// TwinCAT 3 PLC project PlcAppExamples
// Title: PlcAppExamples
// Company: Vortex.Library
// ProjectVersion: 0.6.0.913
// ProgramVersion: 3.1.4024.12
// libraries:
//   Tc2_Standard, * (Beckhoff Automation GmbH)
//   Tc2_System, * (Beckhoff Automation GmbH)
//   Tc3_Module, * (Beckhoff Automation GmbH)
//   TcoCore, 0.6.0.913 (Vortex.Library)
//   TcoPneumatics, 0.6.0.913 (Vortex.Library)
// project tree:
//   / PlcTask.TcTTO
//   POUs/Context/CorleoneKids/ Constanzia_Object.TcPOU, Frederico_Object.TcPOU, Michael_Object.TcPOU, Santino_Object.TcPOU, Thomas_Object.TcPOU
//   POUs/Context/Leaves/ AKid_Object.TcPOU
//   POUs/Context/ VitoCorleone_Context.TcPOU
//   POUs/NonFrameworkUse/ NF_Logic.TcPOU, NF_MAIN.TcPOU
//   POUs/Object/ Horse_Object.TcPOU, Killer_Object.TcPOU, Woltz_Object.TcPOU, Person_Object.TcPOU
//   POUs/Sequencer/ fbAwait.TcPOU, MakeAnOfferThatCantBeRefused.TcPOU, ST_01_Components.TcPOU, ST_01_Context.TcPOU, ST_01_Ground.TcPOU, ST_01_Automat.TcPOU, ST_01_IO.TcGVL
//   POUs/Task/ AskForTheFavor_Task.TcPOU, Kill_Task.TcPOU
//   POUs/Tutorial/101_Color_Sequencer/ ColorSequencer.TcPOU, Color_Example.TcPOU, stColors.TcDUT
//   POUs/Tutorial/201/ InvokingTasks.TcPOU
//   POUs/Tutorial/301/ FastCounter.TcPOU, SlowCounter.TcPOU, TaskExecution.TcPOU
//   POUs/Tutorial/401/ fbPiston.TcPOU, fbPistonMoveTask.TcPOU, IPistonGripper.TcIO, IPistonHorizontal.TcIO, IPistonVertical.TcIO
//   POUs/Tutorial/401/POUs/ Station001.TcPOU, Station001_Components.TcPOU, Station001_Sequencer.TcPOU
//   POUs/Tutorial/ MAIN_PRG.TcPOU, TcOpenTutorial.TcPOU
// real-time tasks:
//   TASK PlcTask: cycle T#10ms, priority 20, ADS port 350

CONFIGURATION PlcAppExamples
    RESOURCE PLC ON TwinCAT3
        TASK PlcTask(INTERVAL := T#10ms, PRIORITY := 20);
        PROGRAM MAIN_PRG WITH PlcTask : MAIN_PRG;
        PROGRAM NF_MAIN WITH PlcTask : NF_MAIN;
    END_RESOURCE
END_CONFIGURATION

// ---- POUs/Tutorial/101_Color_Sequencer/stColors.TcDUT
TYPE stColors :
STRUCT
    _lightR_IsOn : BOOL;
    _lightG_IsOn : BOOL;
    _lightB_IsOn : BOOL;
    _lightR_SwitchOn : BOOL;
    _lightG_SwitchOn : BOOL;
    _lightB_SwitchOn : BOOL;
    _luminosityMin : REAL;
    _luminosity : REAL;
    _luminosityMax : REAL;
END_STRUCT
END_TYPE

// ---- POUs/Sequencer/ST_01_IO.TcGVL
{attribute 'qualified_only'}
VAR_GLOBAL
    INs AT %I* : ARRAY[0..15] OF BOOL;
    OUTs AT %Q* : ARRAY[0..15] OF BOOL;
END_VAR

// ---- POUs/Tutorial/401/IPistonGripper.TcIO
INTERFACE IPistonGripper

METHOD Close : TcoCore.ITcoTaskStatus
END_METHOD

METHOD Open : TcoCore.ITcoTaskStatus
END_METHOD

END_INTERFACE

// ---- POUs/Tutorial/401/IPistonHorizontal.TcIO
INTERFACE IPistonHorizontal

METHOD MoveLeft : TcoCore.ITcoTaskStatus
END_METHOD

METHOD MoveRight : TcoCore.ITcoTaskStatus
END_METHOD

END_INTERFACE

// ---- POUs/Tutorial/401/IPistonVertical.TcIO
INTERFACE IPistonVertical

METHOD MoveDown : TcoCore.ITcoTaskStatus
END_METHOD

METHOD MoveUp : TcoCore.ITcoTaskStatus
END_METHOD

END_INTERFACE

// ---- POUs/Tutorial/MAIN_PRG.TcPOU
PROGRAM MAIN_PRG
VAR
    _pneuMan : ST_01_Context;
    _donCorleone : VitoCorleone_Context;
    _Jack_Woltz : Woltz_Object(_Jack_Woltz);
    _TcOpenTutorial : TcOpenTutorial;
END_VAR

_pneuMan.Run();
_donCorleone.Run();
_TcOpenTutorial.Run();

END_PROGRAM

// ---- POUs/Sequencer/ST_01_Context.TcPOU
// This is an example of a simple pneumatic manipulator 2 pistons 1 gripper.
// Note that this block is extended by 'TcoCore.TcoContext'.
FUNCTION_BLOCK ST_01_Context EXTENDS TcoCore.TcoContext
VAR
    // Ground position sequence
    _groundSequcence : ST_01_Ground(THIS^, eRestoreMode.None);
    // Automat mode sequence
    _automatSequence : ST_01_Automat(THIS^, eRestoreMode.None);
    // Task to execute _groundSequence
    _groundTask : TcoCore.TcoTask(THIS^);
    // Task to execute _automatSequence
    _automatTask : TcoCore.TcoTask(THIS^);
END_VAR

(*~
    <docu>
        <summary>
            Main method of the TcoContext. This is the entry point of any control logic that belongs to this context.
            The call of this method is ensured by calling the <c>InstanceName.Run()</c> method, and it must not be called explicitly.
            This method is abstract, and it must be overriden in inherited block.
        </summary>
    </docu>
~*)
METHOD PROTECTED Main
IF (_groundTask.Execute()) THEN
    _groundSequcence.Run();
    _groundTask.DoneWhen(_groundSequcence._currentStep.ID = 400);
END_IF;

IF (_groundSequcence._currentStep.ID = 400 AND_THEN _automatTask.Execute()) THEN
    _automatSequence.Run();
END_IF;
END_METHOD

END_FUNCTION_BLOCK

// ---- POUs/Sequencer/ST_01_Ground.TcPOU
FUNCTION_BLOCK ST_01_Ground EXTENDS TcoCore.TcoSequencer
VAR
    _components : ST_01_Components(THIS^);
    _await : fbAwait;
END_VAR

(*~
    <docu>
        <summary>
            Main method of the sequener. Custom code needs to be placed here, calling of the methods Open() at the beggining and Close() at the end is ensured by calling the InstanceName.Run() method.
            This method is abstract, so each derived type has to implement its own implementation of this method.
        </summary>
    </docu>
~*)
METHOD PROTECTED Main : BOOL
IF (Step(inStepID := 100, inEnabled := TRUE, inStepDescription := 'VERTICAL CYLINDER UP')) THEN
    //-------------------------------------------------------------
    THIS^.StepCompleteWhen(THIS^._components._vertical.MoveToHome().Done OR _await.Sometime());
    //-------------------------------------------------------------
END_IF

IF (Step(inStepID := 200, inEnabled := TRUE, inStepDescription := 'HORIZONTAL CYLINDER HOME')) THEN
    //-------------------------------------------------------------
    THIS^.StepCompleteWhen(THIS^._components._horizontal.MoveToHome().Done OR _await.Sometime());
    //-------------------------------------------------------------
END_IF

IF (Step(inStepID := 300, inEnabled := TRUE, inStepDescription := 'OPEN GRIPPER')) THEN
    //-------------------------------------------------------------
    THIS^.StepCompleteWhen(THIS^._components._gripper.MoveToHome().Done OR _await.Sometime());
    //-------------------------------------------------------------
END_IF

IF (Step(inStepID := 400, inEnabled := TRUE, inStepDescription := 'CLOSE SEQUENCE')) THEN
    //-------------------------------------------------------------
    //-------------------------------------------------------------
END_IF
END_METHOD

END_FUNCTION_BLOCK

// ---- POUs/Sequencer/ST_01_Components.TcPOU
FUNCTION_BLOCK ST_01_Components EXTENDS TcoCore.TcoObject
VAR
    _horizontal : TcoPneumatics.TcoCylinder(THIS^);
    _vertical : TcoPneumatics.TcoCylinder(THIS^);
    _gripper : TcoPneumatics.TcoCylinder(THIS^);
END_VAR

_horizontal(inoAtHomePos := ST_01_IO.INs[0],
    inoAtWorkPos := ST_01_IO.INs[1],
    inoToHomePos := ST_01_IO.OUTs[0],
    inoToWorkPos := ST_01_IO.OUTs[1]);

_vertical(inoAtHomePos := ST_01_IO.INs[2],
    inoAtWorkPos := ST_01_IO.INs[3],
    inoToHomePos := ST_01_IO.OUTs[2],
    inoToWorkPos := ST_01_IO.OUTs[3]);

_gripper(inoAtHomePos := ST_01_IO.INs[4],
    inoAtWorkPos := ST_01_IO.INs[5],
    inoToHomePos := ST_01_IO.OUTs[4],
    inoToWorkPos := ST_01_IO.OUTs[5]);

END_FUNCTION_BLOCK

// ---- POUs/Sequencer/fbAwait.TcPOU
FUNCTION_BLOCK fbAwait
VAR
    Timer : Tc2_Standard.TON;
END_VAR

METHOD Delay : BOOL
VAR_INPUT
    Timespan : TIME;
END_VAR
Timer(IN := TRUE, PT := Timespan);

IF Timer.Q THEN
    Timer(IN := FALSE, PT := T#0S);
    Delay := TRUE;
ELSE
    Delay := FALSE;
END_IF
END_METHOD

METHOD Sometime : BOOL
VAR_INPUT
END_VAR
Sometime := Delay(T#1S);
END_METHOD

END_FUNCTION_BLOCK

// ---- POUs/Sequencer/ST_01_Automat.TcPOU
FUNCTION_BLOCK ST_01_Automat EXTENDS TcoCore.TcoSequencer
VAR
    _components : ST_01_Components(THIS^);
    _await : fbAwait;
END_VAR

(*~
    <docu>
        <summary>
            Main method of the sequener. Custom code needs to be placed here, calling of the methods Open() at the beggining and Close() at the end is ensured by calling the InstanceName.Run() method.
            This method is abstract, so each derived type has to implement its own implementation of this method.
        </summary>
    </docu>
~*)
METHOD PROTECTED Main : BOOL
_components();

IF (Step(inStepID := 100, inEnabled := TRUE, inStepDescription := 'GROUND')) THEN
    //-------------------------------------------------------------
    THIS^.StepCompleteWhen(_await.Sometime() OR
            (THIS^._components._vertical.MoveToHome().Done AND_THEN
            THIS^._components._horizontal.MoveToHome().Done AND_THEN
            THIS^._components._gripper.MoveToHome().Done));
    //-------------------------------------------------------------
END_IF

IF (Step(inStepID := 200, inEnabled := TRUE, inStepDescription := 'VERTICAL CYLINDER DOWN TO LOAD')) THEN
    //-------------------------------------------------------------
    THIS^.StepCompleteWhen(_await.Sometime() OR (THIS^._components._vertical.MoveToWork().Done));
    //-------------------------------------------------------------
END_IF

IF (Step(inStepID := 300, inEnabled := TRUE, inStepDescription := 'CLOSE GRIPPER')) THEN
    //-------------------------------------------------------------
    THIS^.StepCompleteWhen(_await.Sometime() OR (THIS^._components._gripper.MoveToWork().Done));
    //-------------------------------------------------------------
END_IF

IF (Step(inStepID := 400, inEnabled := TRUE, inStepDescription := 'VERTICAL CYLINDER UP')) THEN
    //-------------------------------------------------------------
    THIS^.StepCompleteWhen(_await.Sometime() OR (THIS^._components._vertical.MoveToHome().Done));
    //-------------------------------------------------------------
END_IF

IF (Step(inStepID := 500, inEnabled := TRUE, inStepDescription := 'HORIZONTAL TO UNLOAD POSITION')) THEN
    //-------------------------------------------------------------
    THIS^.StepCompleteWhen(_await.Sometime() OR (THIS^._components._horizontal.MoveToWork().Done));
    //-------------------------------------------------------------
END_IF

IF (Step(inStepID := 600, inEnabled := TRUE, inStepDescription := 'VERTICAL DOWN TO UNLOAD POSITION')) THEN
    //-------------------------------------------------------------
    THIS^.StepCompleteWhen(_await.Sometime() OR (THIS^._components._vertical.MoveToWork().Done));
    //-------------------------------------------------------------
END_IF

IF (Step(inStepID := 700, inEnabled := TRUE, inStepDescription := 'OPEN GRIPPER')) THEN
    //-------------------------------------------------------------
    THIS^.StepCompleteWhen(_await.Sometime() OR (THIS^._components._gripper.MoveToHome().Done));
    //-------------------------------------------------------------
END_IF

IF (Step(inStepID := 800, inEnabled := TRUE, inStepDescription := 'DONE')) THEN
    //-------------------------------------------------------------
    CompleteSequence();
    //-------------------------------------------------------------
END_IF
END_METHOD

END_FUNCTION_BLOCK

// ---- POUs/Context/VitoCorleone_Context.TcPOU
//--
// <ContextExampleDeclarations>
(*

    THIS EXAMPLE AIMS TO EXPLAIN WHAT CONTEXT AND IDENITY ARE IN A 'TcoOpen' APPLICATION.
    SEE Main() method of this block.

*)
FUNCTION_BLOCK VitoCorleone_Context EXTENDS TcoCore.TcoContext
VAR
    (*
    Each context member object has it 'context' and assigned when instantiated (at birth)
    This is typically done by instantiating the objects with FB_init(ITcoObject) as follows
    These are Don Corleone's children. When you look inside definitions you' find
    Don Corleone's grand-childrend (whole family shares the same context).
*)
    _santino : Santino_Object(THIS^);
    _thomas : Thomas_Object(THIS^);
    _frederico : Frederico_Object(THIS^);
    _michael : Michael_Object(THIS^);
    _costanzia : Constanzia_Object(THIS^);
END_VAR
VAR
    _donCorleoneContext : ITcoContext;
    _isSameContext : BOOL;
    _donCorleoneIdentity : ULINT;
    _isDifferentIndentity : BOOL;
END_VAR
// </ContextExampleDeclarations>
//--
VAR
    _JohnyFontaneCaseDone : BOOL := FALSE;
    _MakeAnOfferThatCantBeRefused : MakeAnOfferThatCantBeRefused(THIS^, eRestoreMode.None);
END_VAR

METHOD JohnyFontaneCase
VAR_INPUT
    Jack_Woltz : REFERENCE TO Woltz_Object;
END_VAR
IF NOT _JohnyFontaneCaseDone THEN
    _MakeAnOfferThatCantBeRefused(Thomas := _thomas, Jack_Woltz := Jack_Woltz, Done => _JohnyFontaneCaseDone);
END_IF;
END_METHOD

(*~
    <docu>
        <summary>
            Main method of the TcoContext. This is the entry point of any control logic that belongs to this context.
            The call of this method is ensured by calling the <c>InstanceName.Run()</c> method, and it must not be called explicitly.
            This method is abstract, and it must be overridden in derived block.
        </summary>
    </docu>
~*)
METHOD PROTECTED Main
//--
// <ContextExampleCode>
(*

                    CONTEXT vs IDENTITY

*)
// In Corleone family they all share the same context that is that of Don Vito Corleone
// Here is the tree of family Corleone
// https://godfather.fandom.com/wiki/Corleone_family
_donCorleoneContext := THIS^.Context;

_isSameContext :=
// Santino
    _donCorleoneContext = THIS^._santino.Context
// Santino's kids
    AND
    (THIS^._santino.Context = THIS^._santino._francesca.Context AND
    THIS^._santino.Context = THIS^._santino._frank.Context AND
    THIS^._santino.Context = THIS^._santino._kathryn.Context AND
    THIS^._santino.Context = THIS^._santino._santino.Context)
// Thomas
    AND
    THIS^._santino.Context = THIS^._thomas.Context
// Thomas' kids
    AND
    (THIS^._thomas.Context = THIS^._thomas._andrew.Context AND
    THIS^._thomas.Context = THIS^._thomas._christina.Context AND
    THIS^._thomas.Context = THIS^._thomas._frank.Context AND
    THIS^._thomas.Context = THIS^._thomas._gianna.Context)
// Frederico
    AND
    THIS^._thomas.Context = THIS^._frederico.Context
// Frederico's kids
    AND
    (THIS^._frederico.Context = THIS^._frederico._fredo.Context)
// Michael
    AND
    THIS^._frederico.Context = THIS^._michael.Context
// Michael's kids
    AND
    (THIS^._michael.Context = THIS^._michael._anthony.Context AND THIS^._michael.Context = THIS^._michael._mary.Context)
// Constanzia
    AND
    THIS^._michael.Context = THIS^._costanzia.Context
// Constanzia's kids
    AND
    (THIS^._costanzia.Context = THIS^._costanzia._michael.Context AND THIS^._costanzia.Context = THIS^._costanzia._victor.Context);
// However each member of the family has different personal identity and that might
// be source of trouble
_donCorleoneIdentity := THIS^.Identity;

_isDifferentIndentity :=
// Santino
    _donCorleoneIdentity <> THIS^._santino.Identity
// Santino's kids
    AND
    (THIS^._santino.Identity <> THIS^._santino._francesca.Identity AND
    THIS^._santino.Identity <> THIS^._santino._frank.Identity AND
    THIS^._santino.Identity <> THIS^._santino._kathryn.Identity AND
    THIS^._santino.Identity <> THIS^._santino._santino.Identity)
// Thomas
    AND
    THIS^._santino.Identity <> THIS^._thomas.Identity
// Thomas' kids
    AND
    (THIS^._thomas.Identity <> THIS^._thomas._andrew.Identity AND
    THIS^._thomas.Identity <> THIS^._thomas._christina.Identity AND
    THIS^._thomas.Identity <> THIS^._thomas._frank.Identity AND
    THIS^._thomas.Identity <> THIS^._thomas._gianna.Identity)
// Frederico
    AND
    THIS^._thomas.Identity <> THIS^._frederico.Identity
// Frederico's kids
    AND
    (THIS^._frederico.Identity <> THIS^._frederico._fredo.Identity)
// Michael
    AND
    THIS^._frederico.Identity <> THIS^._michael.Identity
// Michael's kids
    AND
    (THIS^._michael.Identity <> THIS^._michael._anthony.Identity AND THIS^._michael.Identity <> THIS^._michael._mary.Identity)
// Constanzia
    AND
    THIS^._michael.Identity <> THIS^._costanzia.Identity
// Constanzia's kids
    AND
    (THIS^._costanzia.Identity <> THIS^._costanzia._michael.Identity AND THIS^._costanzia.Identity <> THIS^._costanzia._victor.Identity);
// Once the context is asigned (at birth [instantiated]) it cannot be changed,
// an attempt to change the context will result in vendetta.
// </ContextExampleCode>
//--
JohnyFontaneCase(MAIN_PRG._Jack_Woltz);
END_METHOD

END_FUNCTION_BLOCK

// ---- POUs/Context/CorleoneKids/Santino_Object.TcPOU
FUNCTION_BLOCK Santino_Object EXTENDS TcoCore.TcoObject
VAR
    _francesca : AKid_Object(THIS^);
    _kathryn : AKid_Object(THIS^);
    _frank : AKid_Object(THIS^);
    _santino : AKid_Object(THIS^);
END_VAR

END_FUNCTION_BLOCK

// ---- POUs/Context/Leaves/AKid_Object.TcPOU
FUNCTION_BLOCK AKid_Object EXTENDS TcoCore.TcoObject

END_FUNCTION_BLOCK

// ---- POUs/Context/CorleoneKids/Thomas_Object.TcPOU
FUNCTION_BLOCK Thomas_Object EXTENDS TcoCore.TcoObject
VAR
    _frank : AKid_Object(THIS^);
    _andrew : AKid_Object(THIS^);
    _christina : AKid_Object(THIS^);
    _gianna : AKid_Object(THIS^);
END_VAR
VAR
    _AskForTheFavor : AskForTheFavor_Task(THIS^);
END_VAR

METHOD AskForTheFavor : TcoCore.ITcoTask
VAR_INPUT
    Person_Requested : REFERENCE TO Person_Object;
    RequestedFavor : STRING;
    ReturnFavor : STRING;
END_VAR
_AskForTheFavor(_Person_Requested := Person_Requested, _RequestedFavor := RequestedFavor, _ReturnFavor := ReturnFavor);
AskForTheFavor := _AskForTheFavor;
END_METHOD

END_FUNCTION_BLOCK

// ---- POUs/Task/AskForTheFavor_Task.TcPOU
//--
// <TaskExampleDeclarations>
(*

    This example shows using the 'Tcotask' application. 'TcoTask' is the simplest
    'TcoOpen' coordination primitive.
    In general the body of the task could be devided into the three section:
        1.)	Action
        2.)	Termination condition for the expected behavior.
        3.)	Termination condition for the non-expected behavior.
    The body of the 'Tcotask' needs to be called cyclically. The 'Tcotask' could be then
    invoked from 'outside'. The task of this 'Tcotask' is to ask for the favor
    (in the name of the 'TcoContext' in this example Don Corleone) and offer the return favor.
    Task could end up the expected way in the 'DONE' state if the requested person grant
    the favor or it could end up in the 'ERROR' state if the requested person refuses to grant
    the favor. Each task could be invoked only from the 'READY' state. So if the task enters
    the 'ERROR' state, it cannot be invoked again and has to be restored before. Anyway in this
    example this task is never restored and invoked again as Don Corleone never asks for the
    next favor if the first one was refused.

*)
FUNCTION_BLOCK AskForTheFavor_Task EXTENDS TcoCore.TcoTask
VAR_INPUT
    (*
    'Parameters' of this task are assigned in this example from 'outside' from the
    'upper level' of the hierarchy, where Invoke() method is triggered.
*)
    _Person_Requested : REFERENCE TO Person_Object;
    _RequestedFavor : STRING;
    _ReturnFavor : STRING;
END_VAR
// </TaskExampleDeclarations>
//--

//--
// <TaskBodyExampleCode>
// THIS part needs to be called cyclically.
IF Execute() THEN
    // First section: Action.
    // Meet the right person and interpret the requirements so as a possible return favor.
    _Person_Requested.RequestForTheFavor(_RequestedFavor, _ReturnFavor);
    // Let the person requested to think carefully about the proposition.
    _Person_Requested.ThinkCarefully();
    // Second section: Termination condition for the expected behavior.
    // In the case that the requested person is "smart" and "show the respect" to the
    // 'TcoContext', task finishes in the 'DONE' state and process of the granted the
    // return favor should be started.
    DoneWhen(_Person_Requested.FavorIsGranted());
    // Third section: Termination condition for the non-expected behavior.
    // In the case that the requested person is so self-confident and refuse to grant
    // the favor, task finishes in the 'ERROR' state and automatically the OnTaskError()
    // method is triggered. In this method normally the value of the ReturnFavor is
    // drammatically decreased OR changed to 'Nothing'. Anyway the requested person still
    // have the possibility to grant the favor but under different condition, as he
    // "had to do it the hard way".
    ThrowWhen(_Person_Requested.FavorIsRefused());
END_IF

// </TaskBodyExampleCode>
//--

METHOD PROTECTED OnTaskError
_Person_Requested.ReturnFavor := 'Nothing, and all expenses paid by the recipient.';
END_METHOD

END_FUNCTION_BLOCK

// ---- POUs/Object/Person_Object.TcPOU
FUNCTION_BLOCK Person_Object EXTENDS TcoCore.TcoObject
VAR
    _RequestedFavor : STRING;
    _ReturnFavor : STRING;
    _refuseFavor : BOOL := FALSE;
    _grantFavor : BOOL := FALSE;
END_VAR

METHOD FavorIsGranted : BOOL
VAR_INPUT
END_VAR
FavorIsGranted := _grantFavor;
END_METHOD

METHOD FavorIsRefused : BOOL
VAR_INPUT
END_VAR
FavorIsRefused := _refuseFavor;
END_METHOD

PROPERTY RequestedFavor : String
GET
RequestedFavor := _RequestedFavor;
END_GET
SET
_RequestedFavor := RequestedFavor;
END_SET
END_PROPERTY

METHOD RequestForTheFavor
VAR_INPUT
    inRequestedFavor : STRING;
    inReturnFavor : STRING;
END_VAR
RequestedFavor := inRequestedFavor;
ReturnFavor := inReturnFavor;
END_METHOD

PROPERTY ReturnFavor : String
GET
ReturnFavor := _ReturnFavor;
END_GET
SET
_ReturnFavor := ReturnFavor;
END_SET
END_PROPERTY

METHOD ThinkCarefully
END_METHOD

END_FUNCTION_BLOCK

// ---- POUs/Context/CorleoneKids/Frederico_Object.TcPOU
FUNCTION_BLOCK Frederico_Object EXTENDS TcoCore.TcoObject
VAR
    _fredo : AKid_Object(THIS^);
END_VAR

END_FUNCTION_BLOCK

// ---- POUs/Context/CorleoneKids/Michael_Object.TcPOU
FUNCTION_BLOCK Michael_Object EXTENDS TcoCore.TcoObject
VAR
    _anthony : AKid_Object(THIS^);
    _mary : AKid_Object(THIS^);
END_VAR

END_FUNCTION_BLOCK

// ---- POUs/Context/CorleoneKids/Constanzia_Object.TcPOU
FUNCTION_BLOCK Constanzia_Object EXTENDS TcoCore.TcoObject
VAR
    _victor : AKid_Object(THIS^);
    _michael : AKid_Object(THIS^);
END_VAR

END_FUNCTION_BLOCK

// ---- POUs/Sequencer/MakeAnOfferThatCantBeRefused.TcPOU
FUNCTION_BLOCK MakeAnOfferThatCantBeRefused EXTENDS TcoCore.TcoSequencer
VAR_INPUT
    Thomas : REFERENCE TO Thomas_Object;
    Jack_Woltz : REFERENCE TO Woltz_Object;
END_VAR
VAR_OUTPUT
    Done : BOOL;
END_VAR
VAR
    _FirstOfferAccepted : BOOL := FALSE;
    _FirstOfferRefused : BOOL := FALSE;
    {attribute 'hide'}
    _Killer : Killer_Object(THIS^);
END_VAR

THIS^.Run();

(*~
    <docu>
        <summary>
            Main method of the sequener. Custom code needs to be placed here. The sequencer is executed by call of InstanceName.Run() method.
            This method is abstract, and it must be overridden in derived block.
        </summary>
    </docu>
~*)
METHOD PROTECTED Main : BOOL
IF Step(0, TRUE, 'Send Thomas to ask Jack Woltz for granting the movie role.') THEN
    Done := FALSE;
    // <TaskExternalUseExample>
    //Starting the execution of the 'TcoTask' instance extended by input parameters from 'outside' of the instance.
    Thomas.AskForTheFavor(Jack_Woltz, 'Grant movie role to Johny Fontane.', 'No future problems with unions.').Invoke();
    // Checking from the 'outside' of the instance, if the task has already finished in expected way.
    _FirstOfferAccepted := Thomas._AskForTheFavor.Done;
    // Checking from the 'outside' of the instance, if the task has finished in non-expected way.
    _FirstOfferRefused := Thomas._AskForTheFavor.Error;
    // </TaskExternalUseExample>
    StepCompleteWhen(_FirstOfferAccepted OR _FirstOfferRefused);
END_IF

IF Step(10, _FirstOfferAccepted, 'Call somebody to call somebody to ensure no problems with unions in the future.') THEN
    //*
    //..
    //NoFutureUnionsProblems implementation
    //..
    //*
    RequestStep(500);
END_IF

IF Step(20, TRUE, 'Call somebody to call somebody to send somebody to kill the Woltz horse Khartoum.') THEN
    StepCompleteWhen(_Killer.Kill(Jack_Woltz._Khartoum).Invoke().Done);
END_IF

IF Step(30, TRUE, 'Waiting for granting the movie role to Johny Fontane by Jack Woltz.') THEN
    Jack_Woltz.ThinkCarefully();
    StepCompleteWhen(Jack_Woltz.FavorIsGranted());
END_IF

IF Step(500, TRUE, 'Final step of the sequence.') THEN
    Done := TRUE;
    CompleteStep();
END_IF
END_METHOD

END_FUNCTION_BLOCK

// ---- POUs/Object/Woltz_Object.TcPOU
FUNCTION_BLOCK Woltz_Object EXTENDS Person_Object
VAR
    _Khartoum : Horse_Object(THIS^);
END_VAR

METHOD ThinkCarefully
IF _Khartoum._isAlive THEN
    _refuseFavor := TRUE;
    _grantFavor := FALSE;
ELSE
    _refuseFavor := FALSE;
    _grantFavor := TRUE;
END_IF;
END_METHOD

END_FUNCTION_BLOCK

// ---- POUs/Object/Horse_Object.TcPOU
FUNCTION_BLOCK Horse_Object EXTENDS TcoCore.TcoObject
VAR_INPUT
END_VAR
VAR_OUTPUT
END_VAR
VAR
    _price : REAL := 600000;
    _isAlive : BOOL := TRUE;
END_VAR

PROPERTY IsAlive : Bool
GET
IsAlive := _isAlive;
END_GET
SET
_isAlive := IsAlive;

IF NOT _isAlive THEN
    _price := 0;
END_IF
END_SET
END_PROPERTY

PROPERTY Price : LREAL
GET
IF _isAlive THEN
    Price := _price;
ELSE
    _price := 0;
    Price := _price;
END_IF
END_GET
SET
IF _isAlive THEN
    _price := Price;
ELSE
    _price := 0;
END_IF
END_SET
END_PROPERTY

END_FUNCTION_BLOCK

// ---- POUs/Object/Killer_Object.TcPOU
FUNCTION_BLOCK Killer_Object EXTENDS Person_Object
VAR_INPUT
END_VAR
VAR_OUTPUT
END_VAR
VAR
    _isAlive : BOOL := TRUE;
    _Kill : Kill_Task(THIS^);
END_VAR

PROPERTY IsAlive : Bool
GET
IsAlive := _isAlive;
END_GET
SET
_isAlive := IsAlive;
END_SET
END_PROPERTY

METHOD Kill : TcoCore.ITcoTask
VAR_INPUT
    _Object2bKilled : REFERENCE TO Horse_Object;
END_VAR
_Kill(_Object2bKilled := _Object2bKilled, _Killer := THIS^);
Kill := _Kill;
END_METHOD

END_FUNCTION_BLOCK

// ---- POUs/Task/Kill_Task.TcPOU
FUNCTION_BLOCK Kill_Task EXTENDS TcoCore.TcoTask
VAR_INPUT
    _Object2bKilled : REFERENCE TO Horse_Object;
    _Killer : REFERENCE TO Killer_Object;
END_VAR
VAR_OUTPUT
END_VAR
VAR
END_VAR

IF Execute() THEN
    Kill(_Object2bKilled);
    DoneWhen(NOT _Object2bKilled.IsAlive);
    ThrowWhen(NOT _Killer.IsAlive AND _Object2bKilled.IsAlive);
END_IF

METHOD Kill
VAR_INPUT
    _Object2bKilled : REFERENCE TO Horse_Object;
END_VAR
_Object2bKilled.IsAlive := FALSE;
END_METHOD

END_FUNCTION_BLOCK

// ---- POUs/Tutorial/TcOpenTutorial.TcPOU
FUNCTION_BLOCK TcOpenTutorial EXTENDS TcoCore.TcoContext
VAR
    ColorExample : Color_Example;
    InvokingTasks : InvokingTasks;
    TaskExecution : TaskExecution;
    Station001 : Station001;
END_VAR

// Use Main method instead of this block.

(*~
    <docu>
        <summary>
            Main method of the TcoContext. This is the entry point of any control logic that belongs to this context.
            The call of this method is ensured by calling the <c>InstanceName.Run()</c> method, and it must not be called explicitly.
            This method is abstract, and it must be overridden in derived block.
        </summary>
    </docu>
~*)
METHOD PROTECTED Main
ColorExample.Run();
InvokingTasks.Run();
TaskExecution.Run();
Station001.Run();
END_METHOD

END_FUNCTION_BLOCK

// ---- POUs/Tutorial/101_Color_Sequencer/Color_Example.TcPOU
FUNCTION_BLOCK Color_Example EXTENDS TcoCore.TcoContext
VAR
    ColorSequencer : ColorSequencer(THIS^, eRestoreMode.AutoRestoreMembers);
    Colors : stColors;
END_VAR

// Use Main method instead of this block.

(*~
    <docu>
        <summary>
            Main method of the TcoContext. This is the entry point of any control logic that belongs to this context.
            The call of this method is ensured by calling the <c>InstanceName.Run()</c> method, and it must not be called explicitly.
            This method is abstract, and it must be overridden in derived block.
        </summary>
    </docu>
~*)
METHOD PROTECTED Main
ColorSequencer(inoColors := Colors);
ColorSequencer.Run();
END_METHOD

END_FUNCTION_BLOCK

// ---- POUs/Tutorial/101_Color_Sequencer/ColorSequencer.TcPOU
FUNCTION_BLOCK ColorSequencer EXTENDS TcoCore.TcoSequencer
VAR_INPUT
    inoColors : REFERENCE TO stColors;
END_VAR

// Use Main method instead of this block.

(*~
    <docu>
        <summary>
            Main method of the sequener. Custom code needs to be placed here. The sequencer is executed by call of InstanceName.Run() method.
            This method is abstract, and it must be overridden in derived block.
        </summary>
    </docu>
~*)
METHOD PROTECTED Main : BOOL
// Step header
IF Step(100, // Step id. Must be unique and must change at runtime.
    TRUE, // Indicates that whether the step should execute.
    'Switch all lights off') THEN // Arbitrary step description (for SCADA/HMI)
    //--------------------------------------------
    // Steps logic statements
    inoColors._lightR_SwitchOn := FALSE;
    inoColors._lightG_SwitchOn := FALSE;
    inoColors._lightB_SwitchOn := FALSE;

    IF (NOT inoColors._lightR_IsOn AND NOT inoColors._lightG_IsOn AND NOT inoColors._lightB_IsOn) THEN
        CompleteStep(); // Completes step and moves to step 200
    END_IF;
    //--------------------------------------------
END_IF;

IF Step(200, TRUE, 'Switch on red light') THEN
    //--------------------------------------------
    inoColors._lightR_SwitchOn := TRUE;

    IF (inoColors._lightR_IsOn) THEN
        CompleteStep();
    END_IF;
    //--------------------------------------------
END_IF;

IF Step(300, TRUE, 'Switch on green light') THEN
    //--------------------------------------------
    inoColors._lightG_SwitchOn := TRUE;

    IF (inoColors._lightG_IsOn) THEN
        CompleteStep();
    END_IF;
    //--------------------------------------------
END_IF;

IF Step(400, TRUE, 'Switch on blue light') THEN
    //--------------------------------------------
    inoColors._lightB_SwitchOn := TRUE;

    IF (inoColors._lightB_IsOn) THEN
        CompleteStep();
    END_IF;
    //--------------------------------------------
END_IF;

IF Step(500, TRUE, 'Check that all light are on') THEN
    //--------------------------------------------
    IF (inoColors._lightR_IsOn AND inoColors._lightG_IsOn AND inoColors._lightG_IsOn) THEN
        CompleteStep();
    ELSE
        RequestStep(200); // Some light(s) is(are) not on, try again from 200
    END_IF;
    //--------------------------------------------
END_IF;

IF Step(600, TRUE, 'Measure luminosity') THEN
    //--------------------------------------------
    IF (inoColors._luminosityMin <= inoColors._luminosity AND inoColors._luminosityMax >= inoColors._luminosity) THEN
        CompleteStep();
    ELSE
        RequestStep(500); // Luminosity is not where it should be; check again if the lights are on.
    END_IF

    //--------------------------------------------
END_IF;

IF Step(800, TRUE, 'Complete sequence') THEN
    //--------------------------------------------
    CompleteSequence(); // Returns to the first step (100) in the sequence.
    //--------------------------------------------
END_IF;
END_METHOD

END_FUNCTION_BLOCK

// ---- POUs/Tutorial/201/InvokingTasks.TcPOU
FUNCTION_BLOCK InvokingTasks EXTENDS TcoCore.TcoContext
VAR
    Cylinder : TcoPneumatics.TcoCylinder(THIS^);
    TriggerHome : BOOL;
    TriggerWork : BOOL;
    //simulate IO
    AtHome : BOOL;
    AtWork : BOOL;
    ToHome : BOOL;
    ToWork : BOOL;
    _simTimerValue : UINT := 500;
    _simTimer : Tc2_Standard.TON;
END_VAR

//Use main method

(*~
    <docu>
        <summary>
            Main method of the TcoContext. This is the entry point of any control logic that belongs to this context.
            The call of this method is ensured by calling the <c>InstanceName.Run()</c> method, and it must not be called explicitly.
            This method is abstract, and it must be overridden in derived block.
        </summary>
    </docu>
~*)
METHOD PROTECTED Main
VAR_INST
    ToHomeTemp : BOOL;
    ToWorkTemp : BOOL;
END_VAR
Cylinder(inoAtHomePos := AtHome,
    inoAtWorkPos := AtWork,
    inoToHomePos := ToHome,
    inoToWorkPos := ToWork);

IF ToWork THEN
    AtHome := FALSE;
    _simTimer(IN := TRUE, PT := UINT_TO_TIME(_simTimerValue * 4));

    IF (_simTimer.Q) THEN
        AtWork := TRUE;
        _simTimer(IN := FALSE, PT := UINT_TO_TIME(0));
        Cylinder.Restore();
    END_IF
END_IF

IF ToHome THEN
    AtWork := FALSE;
    _simTimer(IN := TRUE, PT := UINT_TO_TIME(_simTimerValue * 4));

    IF (_simTimer.Q) THEN
        AtHome := TRUE;
        _simTimer(IN := FALSE, PT := UINT_TO_TIME(0));
        Cylinder.Restore();
    END_IF
END_IF

Cylinder.Service(); //enable manual control
END_METHOD

END_FUNCTION_BLOCK

// ---- POUs/Tutorial/301/TaskExecution.TcPOU
FUNCTION_BLOCK TaskExecution EXTENDS TcoCore.TcoContext
VAR
    FastTask : FastCounter(THIS^);
    SlowTask : SlowCounter(THIS^);
END_VAR

// Use main method instead

(*~
    <docu>
        <summary>
            Main method of the TcoContext. This is the entry point of any control logic that belongs to this context.
            The call of this method is ensured by calling the <c>InstanceName.Run()</c> method, and it must not be called explicitly.
            This method is abstract, and it must be overridden in derived block.
        </summary>
    </docu>
~*)
METHOD PROTECTED Main
SlowTask();
FastTask();
END_METHOD

END_FUNCTION_BLOCK

// ---- POUs/Tutorial/301/FastCounter.TcPOU
FUNCTION_BLOCK FastCounter EXTENDS TcoCore.TcoTask
VAR
    Counter : INT;
    _counterProgressCheck : INT;
    _await : fbAwait;
END_VAR

IF Execute() THEN
    IF _await.Delay(T#50MS) THEN
        Counter := Counter + 1;
        _counterProgressCheck := Counter;
    END_IF

    ThrowWhen(_counterProgressCheck > Counter);
    DoneWhen(Counter = 100);
END_IF

(*~
    <docu>
        <summary>
            Restores this instance to the Ready state. Can be called explicitly or from within one of the restore mechanisms.
            <para>
                See also <see cref="PlcDocu.TcoCore.TcoTask.AutoRestorable()"/>
            </para>
        </summary>
    </docu>
~*)
METHOD Restore : ITcoRestorable
SUPER^.Restore();
Counter := 0;
_counterProgressCheck := 0;
END_METHOD

END_FUNCTION_BLOCK

// ---- POUs/Tutorial/301/SlowCounter.TcPOU
FUNCTION_BLOCK SlowCounter EXTENDS TcoCore.TcoTask
VAR
    Counter : INT;
    _await : fbAwait;
END_VAR

IF Execute() THEN
    IF _await.Delay(T#250MS) THEN
        Counter := Counter + 1;
    END_IF

    DoneWhen(Counter = 100);
END_IF

(*~
    <docu>
        <summary>
            Restores this instance to the Ready state. Can be called explicitly or from within one of the restore mechanisms.
            <para>
                See also <see cref="PlcDocu.TcoCore.TcoTask.AutoRestorable()"/>
            </para>
        </summary>
    </docu>
~*)
METHOD Restore : ITcoRestorable
SUPER^.Restore();
Counter := 0;
END_METHOD

END_FUNCTION_BLOCK

// ---- POUs/Tutorial/401/POUs/Station001.TcPOU
FUNCTION_BLOCK Station001 EXTENDS TcoCore.TcoContext
VAR
    _components : Station001_Components(THIS^);
    _sequence : Station001_Sequencer(THIS^, eRestoreMode.None, _components);
END_VAR

(*~
    <docu>
        <summary>
            Main method of the TcoContext. This is the entry point of any control logic that belongs to this context.
            The call of this method is ensured by calling the <c>InstanceName.Run()</c> method, and it must not be called explicitly.
            This method is abstract, and it must be overridden in derived block.
        </summary>
    </docu>
~*)
METHOD PROTECTED Main
_components();
_sequence.Run();
END_METHOD

END_FUNCTION_BLOCK

// ---- POUs/Tutorial/401/POUs/Station001_Components.TcPOU
FUNCTION_BLOCK Station001_Components EXTENDS TcoCore.TcoObject
VAR
    {attribute addProperty Name "Horizontal cyclinder A1"}
    _horizontal : fbPiston(THIS^);
    {attribute addProperty Name "Vertical cyclinder A2"}
    _vertical : fbPiston(THIS^);
    {attribute addProperty Name "Gripper A3"}
    _gripper : fbPiston(THIS^);
END_VAR
VAR
    _simTimerValue : UINT := 500;
    _simTimer : Tc2_Standard.TON;
END_VAR

_vertical();
_horizontal();
_gripper();
_simTimer(IN := TRUE, PT := UINT_TO_TIME(_simTimerValue));
SimulateCylinder(_vertical);
SimulateCylinder(_horizontal);
SimulateCylinder(_gripper);

PROPERTY Gripper : IPistonGripper
GET
Gripper := _gripper;
END_GET
END_PROPERTY

PROPERTY Horizontal : IPistonHorizontal
GET
Horizontal := _horizontal;
END_GET
END_PROPERTY

METHOD SimulateCylinder
VAR_IN_OUT
    ioCyclinder : fbPiston;
END_VAR
ioCyclinder.iHomePositionSensor := ioCyclinder.qHomePositionActuator AND _simTimer.Q;
ioCyclinder.iWorkPositionSensor := ioCyclinder.qWorkPositionActuator AND _simTimer.Q;
END_METHOD

PROPERTY Vertical : IPistonVertical
GET
Vertical := _vertical;
END_GET
END_PROPERTY

END_FUNCTION_BLOCK

// ---- POUs/Tutorial/401/fbPiston.TcPOU
{attribute addProperty Name "Pneumatic cyclinder"}
FUNCTION_BLOCK fbPiston EXTENDS TcoCore.TcoComponent IMPLEMENTS IPistonGripper, IPistonHorizontal, IPistonVertical
VAR_INPUT
    iHomePositionSensor : BOOL;
    iWorkPositionSensor : BOOL;
END_VAR
VAR_OUTPUT
    qHomePositionActuator : BOOL;
    qWorkPositionActuator : BOOL;
END_VAR
VAR
    {attribute addProperty Activity "moves to home position"}
    _moveHomeTask : fbPistonMoveTask(THIS^);
    {attribute addProperty Activity "moves to work position"}
    _moveWorkTask : fbPistonMoveTask(THIS^);
END_VAR

_moveHomeTask(PositionSensor := iHomePositionSensor, MoveToPositionSignal := qHomePositionActuator, InverseSignal := qWorkPositionActuator);
_moveWorkTask(PositionSensor := iWorkPositionSensor, MoveToPositionSignal := qWorkPositionActuator, InverseSignal := qHomePositionActuator);

METHOD Close : TcoCore.ITcoTaskStatus
Close := MoveToHome();
END_METHOD

METHOD PROTECTED Manual
VAR_INPUT
END_VAR
END_METHOD

METHOD MoveDown : TcoCore.ITcoTaskStatus
MoveDown := MoveToHome();
END_METHOD

METHOD MoveLeft : TcoCore.ITcoTaskStatus
MoveLeft := MoveToWork();
END_METHOD

METHOD MoveRight : TcoCore.ITcoTaskStatus
MoveRight := MoveToHome();
END_METHOD

METHOD PROTECTED MoveToHome : TcoCore.ITcoTaskStatus
MoveToHome := THIS^._moveHomeTask.Invoke();
END_METHOD

METHOD PROTECTED MoveToWork : TcoCore.ITcoTaskStatus
MoveToWork := THIS^._moveWorkTask.Invoke();
END_METHOD

METHOD MoveUp : TcoCore.ITcoTaskStatus
MoveUp := MoveToWork();
END_METHOD

METHOD Open : TcoCore.ITcoTaskStatus
Open := MoveToWork();
END_METHOD

METHOD Restore : ITcoRestorable
THIS^._moveHomeTask.Restore();
THIS^._moveWorkTask.Restore();
END_METHOD

(*~
    <docu>
        <summary>
            Custom service (manual, maintenance) logic.
            This method must be implemented in derived class.
        </summary>
    </docu>
~*)
METHOD PROTECTED ServiceMode
END_METHOD

END_FUNCTION_BLOCK

// ---- POUs/Tutorial/401/fbPistonMoveTask.TcPOU
{attribute addProperty Activity "task is running"}
FUNCTION_BLOCK fbPistonMoveTask EXTENDS TcoCore.TcoTask
VAR_INPUT
    PositionSensor : BOOL;
END_VAR
VAR_IN_OUT
    MoveToPositionSignal : BOOL;
    InverseSignal : BOOL;
END_VAR

IF (THIS^.Execute()) THEN
    THIS^.Messenger.Debug('|[[1]AttributeName]| |[AttributeActivity]|, extremity sensor not reached yet.');
    InverseSignal := FALSE;
    MoveToPositionSignal := TRUE;
    THIS^.DoneWhen(PositionSensor);
END_IF

END_FUNCTION_BLOCK

// ---- POUs/Tutorial/401/POUs/Station001_Sequencer.TcPOU
FUNCTION_BLOCK Station001_Sequencer EXTENDS TcoCore.TcoSequencer
VAR
    components : REFERENCE TO Station001_Components;
END_VAR
VAR
    _switchToStep : BOOL;
    _failedToLoad : BOOL;
END_VAR

METHOD FB_init : BOOL
VAR_INPUT
    bInitRetains : BOOL; // if TRUE, the retain variables are initialized (warm start / cold start)
    bInCopyCode : BOOL; // if TRUE, the instance afterwards gets moved into the copy code (online change)
    ParentObject : ITcoObject;
    AutoRestoreMode : eRestoreMode;
    refComponents : REFERENCE TO Station001_Components;
END_VAR
Components REF= refComponents;
END_METHOD

METHOD Init
VAR_INPUT
END_VAR
components();

IF (Step(0, TRUE, 'INIT')) THEN
    //-----------------------------------------------------
    THIS^.StepCompleteWhen(TRUE);
    //-----------------------------------------------------
END_IF
END_METHOD

(*~
    <docu>
        <summary>
            Main method of the sequener. Custom code needs to be placed here. The sequencer is executed by call of InstanceName.Run() method.
            This method is abstract, and it must be overridden in derived block.
        </summary>
    </docu>
~*)
METHOD PROTECTED Main : BOOL
Init();

IF (Step(100, TRUE, 'MOVE ALL CYLINDERS TO GROUND POSITION')) THEN
    //-----------------------------------------------------
    StepCompleteWhen(components.Vertical.MoveUp().Done AND_THEN components.Horizontal.MoveLeft().Done AND_THEN components.Gripper.Open().Done);
    //-----------------------------------------------------
END_IF

IF (Step(200, TRUE, 'MOVE VERTICAL CYLINDER DOWN')) THEN
    //-----------------------------------------------------
    StepCompleteWhen(components.Vertical.MoveDown().Done);
    //-----------------------------------------------------
END_IF

IF (Step(300, TRUE, 'CLOSE GRIPPER')) THEN
    //-----------------------------------------------------
    IF (components.Gripper.Close().Done) THEN
        IF (_failedToLoad) THEN
            RequestStep(100);
        ELSE
            StepCompleteWhen(TRUE);
        END_IF;
    END_IF;
    //-----------------------------------------------------
END_IF

IF (Step(400, TRUE, 'MOVE VERTICAL CYLINDER UP')) THEN
    //-----------------------------------------------------
    StepCompleteWhen(components.Vertical.MoveUp().Done);
    //-----------------------------------------------------
END_IF

IF (Step(500, TRUE, 'MOVE HORIZONTAL CYLINDER TO UNLOAD POSITION')) THEN
    //-----------------------------------------------------
    StepCompleteWhen(components.Horizontal.MoveRight().Done);
    //-----------------------------------------------------
END_IF

IF (Step(600, TRUE, 'MOVE VERTICAL CYLINDER DOWN')) THEN
    //-----------------------------------------------------
    StepCompleteWhen(components.Vertical.MoveDown().Done);
    //-----------------------------------------------------
END_IF

IF (Step(700, TRUE, 'OPEN GRIPPER')) THEN
    //-----------------------------------------------------
    StepCompleteWhen(components.Gripper.Open().Done);
    //-----------------------------------------------------
END_IF

IF (Step(800, TRUE, 'CLOSE SEQUENCE')) THEN
    //-----------------------------------------------------
    CompleteSequence();
    //-----------------------------------------------------
END_IF
END_METHOD

METHOD PROTECTED OnStateChange
VAR_INPUT
    PreviousState : INT;
    NewState : INT;
END_VAR
components._simTimer(IN := FALSE);
END_METHOD

END_FUNCTION_BLOCK

// ---- POUs/NonFrameworkUse/NF_MAIN.TcPOU
PROGRAM NF_MAIN
VAR
    _context : TcoCore.TcoContextNfCompatibility;
    _logic : NF_Logic;
END_VAR

_context.VolatileOpen();
_logic();
_context.VolatileClose();

PROPERTY Context : REFERENCE TO TcoCore.TcoContextNfCompatibility
GET
Context REF= _context;
END_GET
END_PROPERTY

END_PROGRAM

// ---- POUs/NonFrameworkUse/NF_Logic.TcPOU
FUNCTION_BLOCK NF_Logic
VAR
    _piston : TcoPneumatics.TcoCylinder(NF_MAIN.Context);
    _signals : ARRAY[0..3] OF BOOL;
END_VAR

_piston.Service();

_piston(inoAtHomePos := _signals[0],
    inoAtWorkPos := _signals[1],
    inoToHomePos := _signals[2],
    inoToWorkPos := _signals[3]);

END_FUNCTION_BLOCK
